TYPE ST_MotionDrive :
    // Translated into properties and move to EPICS interface.
STRUCT
    test : BOOL;

END_STRUCT
END_TYPE

(* stored: Version 1.1.0.1
   DUT ST_MotionDrive: Id {f4cf3312-62a3-4683-ad20-6d4fcdde1d39} *)
